# B&R Automation Studio project Lib_PathKin
Automation Studio 4.7.3.93 SP

## Configuration ARsim

### Task classes (Cpu.sw)
```

```

## Logical view

Binary libraries used (declarations not repeated): operator, runtime, astime, AsIecCon, PathKin

### Package Logical/Libraries - Global libraries

### Library Logical/Libraries/MathTools (ANSIC) - Miscellaneous math functions

#### MathTools.fun
```iecst
(*Integer wrap*)

FUNCTION Math_WrapUSINT : USINT
	VAR_INPUT
		Value : DINT;
		LowerBound : DINT;
		UpperBound : DINT;
	END_VAR
END_FUNCTION

FUNCTION Math_WrapSINT : SINT
	VAR_INPUT
		Value : DINT;
		LowerBound : DINT;
		UpperBound : DINT;
	END_VAR
END_FUNCTION

FUNCTION Math_WrapUINT : UINT
	VAR_INPUT
		Value : DINT;
		LowerBound : DINT;
		UpperBound : DINT;
	END_VAR
END_FUNCTION

FUNCTION Math_WrapINT : INT
	VAR_INPUT
		Value : DINT;
		LowerBound : DINT;
		UpperBound : DINT;
	END_VAR
END_FUNCTION
(*Floating point wrap*)

FUNCTION Math_WrapREAL : REAL
	VAR_INPUT
		Value : LREAL;
		LowerBound : LREAL;
		UpperBound : LREAL;
	END_VAR
END_FUNCTION

FUNCTION Math_WrapLREAL : LREAL
	VAR_INPUT
		Value : LREAL;
		LowerBound : LREAL;
		UpperBound : LREAL;
	END_VAR
END_FUNCTION
(*Quadtratic formula*)

FUNCTION Math_2ndOrderRoots : BOOL
	VAR_INPUT
		p2 : LREAL;
		p1 : LREAL;
		p0 : LREAL;
	END_VAR
	VAR_IN_OUT
		Solution : Math2ndOrderRootsSoln_typ;
	END_VAR
END_FUNCTION
(*Heaviside function*)

FUNCTION Math_UnitStep : REAL
	VAR_INPUT
		Input : LREAL;
	END_VAR
END_FUNCTION
```

#### math_tools.c
```c
/*********************************************************************************
 * Copyright: B&R Industrial Automation
 * Author:    Tyler Matijevich
 * Created:   May 14, 2020/1:34 PM
 *********************************************************************************/

#include "MathTools.h"
#include <math.h>

/*
 * Internal function
 * Utilize the implicit conversion from chars/shorts to longs
 */
static signed long WrapInteger(signed long inputValue, signed long lowerBound, signed long upperBound) {
	/* Static functions are functions only visible to other functions in the file */

	if(lowerBound <= upperBound) {
		signed long total 		= upperBound - lowerBound + 1;
		signed long distance 	= inputValue - lowerBound;
		signed long offset 		= distance % total;

		if(offset >= 0)
			return lowerBound + offset;
		else
			return upperBound + offset + 1; // +1 to include the upper bound during subtraction
	}

	else
		return 0;

}

/*
 * Each function will return zero if the bounds exceed data type limits
 * or the lower bound exceeds the upper bound
 */

/* USINT wrap */
unsigned char Math_WrapUSINT(signed long Value, signed long LowerBound, signed long UpperBound) {
	if(LowerBound < 0 || LowerBound > 255 || UpperBound < 0 || UpperBound > 255)
		return 0;
	else
		return (unsigned char)WrapInteger(Value, LowerBound, UpperBound);
}

/* SINT wrap */
signed char Math_WrapSINT(signed long Value, signed long LowerBound, signed long UpperBound) {
	if(LowerBound < -128 || LowerBound > 127 || UpperBound < -128 || UpperBound > 127)
		return 0;
	else
		return (signed char)WrapInteger(Value, LowerBound, UpperBound);
}

/* UINT wrap */
unsigned short Math_WrapUINT(signed long Value, signed long LowerBound, signed long UpperBound) {
	if(LowerBound < 0 || LowerBound > 65535 || UpperBound < 0 || UpperBound > 65535)
		return 0;
	else
		return (unsigned short)WrapInteger(Value, LowerBound, UpperBound);
}

/* INT wrap */
signed short Math_WrapINT(signed long Value, signed long LowerBound, signed long UpperBound) {
	if(LowerBound < -32768 || LowerBound > 32767 || UpperBound < -32768 || UpperBound > 32767)
		return 0;
	else
		return (signed short)WrapInteger(Value, LowerBound, UpperBound);
}

/*
 * Internal function
 * Utilize the implicit conversion from floats to doubles
 */
double WrapDouble(double inputValue, double lowerBound, double upperBound) {
	if(upperBound > lowerBound){
		double distance = inputValue - lowerBound;
		double total = upperBound - lowerBound;
		double offset = distance - trunc(distance / total) * total;
		return (distance >= 0.0)? (lowerBound + offset) : (upperBound + offset);
	} else
		return 0.0;
}

/* REAL wrap */
float Math_WrapREAL(double Value, double LowerBound, double UpperBound) {
	return (float)WrapDouble(Value, LowerBound, UpperBound);
}

/* LREAL wrap */
double Math_WrapLREAL(double Value, double LowerBound, double UpperBound) {
	return WrapDouble(Value, LowerBound, UpperBound);
}

/* 2nd Order Roots (Quadratic formula) $$ p2 * x^2 + p1 * x + p0 = 0 $$ */
unsigned char Math_2ndOrderRoots(double p2, double p1, double p0, struct Math2ndOrderRootsSoln_typ* Solution) {
	Solution->r1 = Solution->r2 = 0.0; /* Default/Invalid solution */
	double determinant = pow(p1, 2.0) - 4.0 * p2 * p0;

	if(fabs(p2) > 0.0) { /* Two roots - protect against divide by zero */
		if(determinant > 0.0) {
			Solution->r1 = ((-p1) + sqrt(determinant)) / (2.0 * p2);
			Solution->r2 = ((-p1) - sqrt(determinant)) / (2.0 * p2);
		}

		else if(determinant < 0.0)
			return 11; /* Status Code 11: Imaginary roots, do not consider this case */

		else {
			Solution->r1 = (-p1) / (2.0 * p2);
			Solution->r2 = Solution->r1;
		}
		return 0;

	} else {
		if(fabs(p1) > 0.0) { /* One root - protect against divide by zero */
			Solution->r1 = (-p0) / p1;
			Solution->r2 = Solution->r1;
			return 0;

		} else /* No solution */
			return 12; /* Status Code 12: No solution */
	}
}

/* Heaviside function */
float Math_UnitStep(double Input){
	return (Input >= 0.0)? 1.0 : 0.0;
}
```

### Program Logical/Example

#### Variables.var
```iecst
VAR
	dt : REAL;
	dx : REAL;
	v0 : REAL;
	vf : REAL;
	vmin : REAL;
	vmax : REAL;
END_VAR
(*Kin_GetAcc()*)
VAR
	AccSoln : KinGetAccSoln_typ;
	status_GetAcc : USINT;
END_VAR
(*Kin_GetAccInTimespanPlus()*)
VAR
	AccInTimespanPlusSoln : KinGetAccInTimespanSoln_typ;
	status_GetAccInTimespanPlus : USINT;
END_VAR
(*Kin_GetTimespan()*)
VAR
	TimespanSoln : KinGetTimespanSoln_typ;
	status_GetTimespan : USINT;
END_VAR
(*Kin_GetVelProfPoint()*)
VAR
	times : ARRAY[0..KIN_MAX_PROF_POINTS] OF REAL;
	velocities : ARRAY[0..KIN_MAX_PROF_POINTS] OF REAL;
	VelProfPointSoln : KinGetVelProfPointSoln_typ;
	status_GetVelProfPoint : USINT;
END_VAR
```

#### Main.st
```iecst
(*******************************************************************************
 * Copyright: B&R Industrial Automation
 * Author:    Tyler Matijevich
 * Created:   May 14, 2020/6:28 PM
********************************************************************************
 * Description: Example program to test the PathKin library
********************************************************************************)

PROGRAM _INIT

	dt := 0.300;
	dx := 0.350;
	v0 := 1.9;
	vf := 1.2;
	vmin := 0.75;
	vmax := 3.0;

	times[1] := 0.0;
	times[2] := 0.25;
	times[3] := 0.4;
	times[4] := 0.5;
	times[5] := 0.6;

	velocities[1] := 0.0;
	velocities[2] := 1.9;
	velocities[3] := 0.75;
	velocities[4] := 0.75;
	velocities[5] := 1.2;

END_PROGRAM

PROGRAM _CYCLIC

	status_GetAcc := Kin_GetAcc(dt, dx, v0, vf, vmin, vmax, AccSoln);

	status_GetAccInTimespanPlus := Kin_GetAccInTimespanPlus(dt, dx, v0, vf, vmin, vmax, AccInTimespanPlusSoln);

	status_GetTimespan := Kin_GetTimespan(dx - EXPT(v0, 2) / (2.0 * AccInTimespanPlusSoln.a), v0, vf, vmin, vmax, AccInTimespanPlusSoln.a, TimespanSoln);

	status_GetVelProfPoint := Kin_GetVelProfPoint(0.0, times, velocities, 5, 0.515, VelProfPointSoln);

END_PROGRAM

PROGRAM _EXIT

END_PROGRAM
```

Listed in the project but not available here: Logical/Global.typ, Logical/Global.var
